PROGRAM MAIN
VAR
	
Coordinador : FB_Coordinador_ST;

END_VAR

Coordinador();

END_PROGRAM

(* stored: Version 1.1.0.1, ProductVersion 3.1.4024.11
   POU MAIN: Id {c92b9105-0189-4ab8-bb90-5be8fb337865}, SpecialFunc None *)
